TYPE PLCToHMIOperatingMode :
STRUCT
	Manuel	:	ActionState;
	Automatic	:	ActionState;
	AutomaticStart	:	ActionState;
	Automaticstop	:	ActionState;
	AutomaticHome	:	ActionState;
	Reset	:	ActionState;
	Quit	:	ActionState;
	Fault	:	ActionState;
	
END_STRUCT
END_TYPE

(* stored: Version 1.1.0.1
   DUT PLCToHMIOperatingMode: Id {95cbae51-f4ba-43cf-905a-89be056966bd} *)
